GLOBALCONSTANTS AID_OR (* Output rectangle object attribute ids *)
  (* Standard: 61499-1; Description: Copyright (c) 2023 HR Agrartechnik GmbH This program and the accompanying materials are made available under the terms of the Eclipse Public License 2.0 which is available at https://www.eclipse.org/legal/epl-2.0/ SPDX-License-Identifier: EPL-2.0 *)
  (* Version 1.0, 2026-06-20, Franz Höpfinger, HR Agrartechnik GmbH *)
  PACKAGE isobus::UT::Q::const::AID;
  IMPORT eclipse4diac::core::TypeHash;
  VAR_GLOBAL CONSTANT
    LINE_ATT : USINT := USINT#1; (* 1: AID_OR_LINE_ATT - Object ID of a Line Attributes object. *)
    WIDTH : USINT := USINT#2; (* 2: AID_OR_WIDTH - Width in pixels. *)
    HEIGHT : USINT := USINT#3; (* 3: AID_OR_HEIGHT - Height in pixels. *)
    LINE_SUPPR : USINT := USINT#4; (* 4: AID_OR_LINE_SUPPR *)
    FILL_ATT : USINT := USINT#5; (* 5: AID_OR_FILL_ATT - Object ID of a Fill Attributes object. *)
  END_VAR
END_GLOBALCONSTANTS
